// TIA Portal V17 export
// export: Created 2023-02-13T11:16:52.2273647Z, ExportSetting WithDefaults, DisplayName Totally Integrated Automation Portal, DisplayVersion V17, DisplayName TIA Portal Openness, DisplayVersion V17, DisplayName TIA Portal Teamcenter Gateway, DisplayVersion V17, DisplayName TIA Portal Version Control Interface, DisplayVersion V17, DisplayName SINAMICS Startdrive Advanced, DisplayVersion V17, DisplayName SINAMICS Startdrive G130, G150, S120, S150, SINAMICS MV, S210, DisplayVersion V17, DisplayName SINAMICS Startdrive G110M, G120, G120C, G120D, G120P, G115D, DisplayVersion V17, DisplayName STEP 7 Professional, DisplayVersion V17, DisplayName STEP 7 Safety, DisplayVersion V17, DisplayName WinCC Professional, DisplayVersion V17
FUNCTION_BLOCK "HWT"   // FB350, LAD
{ S7_Optimized_Access := 'TRUE' }
VERSION : 0.1
// stored: AutoNumber false, IsIECCheckEnabled false, IsRetainMemResEnabled false, MemoryReserve 100, SetENOAutomatically false, UDAEnableTagReadback false
   VAR_INPUT
      "IN_FBAV.01" : Bool := FALSE;   // Tank Return Valve
      "IN_FBAV.02" : Bool := FALSE;   // Tank Water Inlet Valve
      "IN_FBAV.03" : Bool := FALSE;   // Tank CIP Return Valve
      "IN_FBAV.04" : Bool := FALSE;   // Tank CIP Inlet Valve
      "IN_FBAV.10" : Bool := FALSE;   // Steam Shutoff Valve
      "IN_FBCV.10" : Bool := FALSE;   // Steam Control Valve
      "IN_FS.01" : Bool := FALSE;   // Line Flow Switch
      IN_LT01 : Real;   // Tank Level Transmitter
      IN_TT01 : Real;   // Tank Temp. Transmitter
      IN_TT02 : Real;   // Line Temp. Transmitter
      "IN_FBP.01" : Bool;   // Hot Water Pump
      "IN_P.01-Speed" : Real := 0.0;   // Hot Water Pump AV Speed
      DosePumpSpeed : Real;
      "DoseON-OFF" : Bool;
      "DosePumpON-OFF" : Bool;
      CIPPulse : Bool;
      Line_OK : Bool;
   END_VAR
   VAR_OUTPUT
      "OUT_AV.01" : Bool := FALSE;   // Tank Return Valve
      "OUT_AV.02" : Bool := FALSE;   // Tank Water Inlet Valve
      "OUT_AV.03" : Bool := FALSE;   // Tank CIP Return Valve
      "OUT_AV.04" : Bool := FALSE;   // Tank CIP Inlet Valve
      "OUT_AV.10" : Bool := FALSE;   // Steam Shutoff Valve
      "OUT_CV.10" : Bool := FALSE;   // Steam Control Valve
      Q_PID_Setpoint : Real;
      Q_PID_PV_IN : Real;
      "OUT_FS.01" : Bool := FALSE;   // Line Flow Switch
      "OUT_LT.01" : Real;   // Tank Level Transmitter
      "OUT_TT.01" : Real;   // Tank Temp. Transmitter
      "OUT_TT.02" : Real;   // Line Temp. Transmitter
      "OUT_P.01" : Bool := FALSE;   // Hot Water Pump
      "OUT_P.01-Speed" : Real := 0.0;   // Hot Water Pump SP Speed
      OUT_CIP_Request : Bool;
      Q_WH_Tank_Ready : Bool;
   END_VAR
   VAR
      Cmd : Struct
         Start_Prosses : Bool;
         Start_Preheat : Bool;
         HWT_Mode : Bool;
         Ready_for_Mix : Bool;
         "CIP Request" : Bool;
         Pump_Mode : Bool;
         Pump_Man_ON_OFF : Bool;
      END_STRUCT;
      Param : Struct
         SP_Level_LL : Real := 10.0;
         SP_Level_ML : Real := 80.0;
         SP_Level_HL : Real := 100.0;
         SP_Temp_Prepar : Real := 80.0;
         SP_Temp_Process : Real := 80.0;
         SP_PumpSpeed : Real := 80.0;
         L_Hi_Lim : Real := 100.0;
         L_Lo_Lim : Real := 0.0;
         L_Hys : Real := 5.0;
         T_Hi_Lim : Real := 100.0;
         T_Lo_Lim : Real := 0.0;
         T_Hys : Real := 2.0;
         CIP_Ret_ON_SP : Real := 5.0;
         CIP_Ret_OFF_SP : Real;
      END_STRUCT;
      State : Struct
         Tank_LL : Bool;
         Tank_ML : Bool;
         Tank_HL : Bool;
         Temp_Preheat_OK : Bool;
         Temp_Process_OK : Bool;
         Tank_Heating : Bool;
         "Tank is Ready" : Bool;
         "Tank in transfer" : Bool;
         Enable_WHT_Mode : Bool;
         Enable_Ready : Bool;
         Ready_for_Mix : Bool;
         "CIP Request Enable" : Bool;
         "Tank in CIP" : Bool;
         CIP_Request_OK : Bool;
         CIP_ReturnON : Bool;
         HWT_Status : Int;
         Temp_Actual : Real;
      END_STRUCT;
      L_Hys_Abs : Real;
      T_Hys_Abs : Real;
      Hys_Level_HL : Real;
      Hys_Level_ML : Real;
      Hys_Level_LL : Real;
      "Hys SP_SP_Prepar" : Real;
      "Hys SP_SP_Process" : Real;
      "Hys SP_SP_" : Real;
      alwaysON : Bool;
      r : Struct
         PosE1 : Bool;
         PosE2 : Bool;
         PosE3 : Bool;
         PosE4 : Bool;
         PosE5 : Bool;
         PosE6 : Bool;
         PosE7 : Bool;
         PosE8 : Bool;
         PosE9 : Bool;
         PosE10 : Bool;
         PosE11 : Bool;
         PosE12 : Bool;
         PosE13 : Bool;
         PosE14 : Bool;
         PosE15 : Bool;
         PosE16 : Bool;
         PosE17 : Bool;
         PosE18 : Bool;
         PosE19 : Bool;
         PosE20 : Bool;
         PosE21 : Bool;
         PosE22 : Bool;
         PosE23 : Bool;
         PosE24 : Bool;
         PosE25 : Bool;
         PosE26 : Bool;
         PosE27 : Bool;
         PosE28 : Bool;
         PosE29 : Bool;
         PosE30 : Bool;
         PosE31 : Bool;
         PosE32 : Bool;
      END_STRUCT;
      Actuator : Struct
         AV_Inlet : Bool;
         AV_Return : Bool;
         CV_Steam : Bool;
         Pump : Bool;
      END_STRUCT;
      r_Pump : Bool;
      r_PumpTim { S7_SetPoint := 'True'} : IEC_TIMER;
      Alarm : Word;
      Event : Word;
   END_VAR
   VAR_TEMP   // added for the SCL form of the ladder/FBD networks
      _w1 : Bool;
      _w2 : Bool;
   END_VAR
BEGIN

REGION Network 1: Always_ON
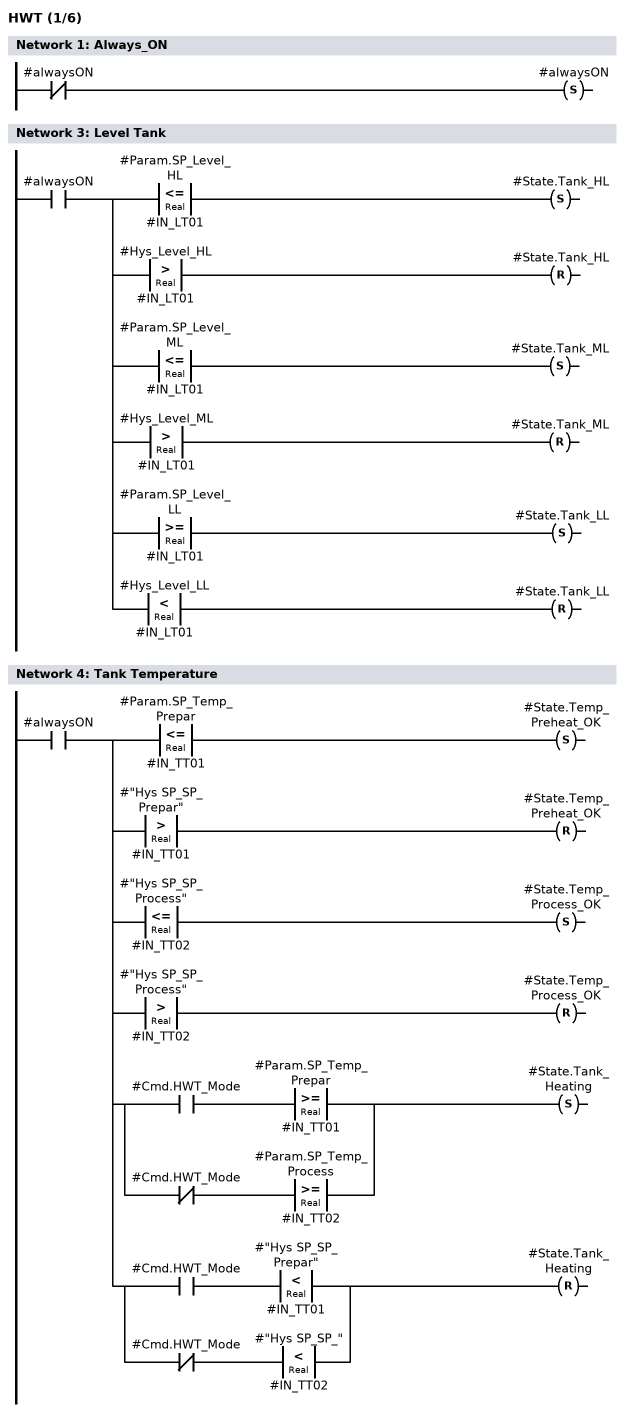
   RUNG wire#powerrail
      I_Contact( #alwaysON )
      S_Coil( #alwaysON )
   END_RUNG
   // the same network as SCL:
   IF NOT #alwaysON THEN #alwaysON := TRUE; END_IF;
END_REGION

NETWORK
TITLE = Hys Calculation
//Level Hys Absolute
      L     #Param.L_Hi_Lim;
      L     #Param.L_Lo_Lim;
      -R;
      L     100.0;
      /R;
      L     #Param.L_Hys;
      *R;
      T     #L_Hys_Abs;
//Temp. Hys Absolute
      L     #Param.T_Hi_Lim;
      L     #Param.T_Lo_Lim;
      -R;
      L     100.0;
      /R;
      L     #Param.T_Hys;
      *R;
      T     #T_Hys_Abs;
//Tank High Level
      L     #Param.SP_Level_HL;
      L     #L_Hys_Abs;
      -R;
      T     #Hys_Level_HL;
//Tank Mid Level
      L     #Param.SP_Level_ML;
      L     #L_Hys_Abs;
      -R;
      T     #Hys_Level_ML;
//Tank Low Level
      L     #Param.SP_Level_LL;
      L     #L_Hys_Abs;
      +R;
      T     #Hys_Level_LL;
//Temp. Preheat Hys
      L     #Param.SP_Temp_Prepar;
      L     #T_Hys_Abs;
      +R;
      T     #"Hys SP_SP_Prepar";
//Temp. Transfer Hys
      L     #Param.SP_Temp_Process;
      L     #T_Hys_Abs;
      -R;
      T     #"Hys SP_SP_Process";
//Temp. Transfer Heating Hys
      L     #Param.SP_Temp_Process;
      L     #T_Hys_Abs;
      +R;
      T     #"Hys SP_SP_";


REGION Network 3: Level Tank
   RUNG wire#powerrail
      Contact( #alwaysON )
      wire#w1
      { S7_Templates := "SrcType := Real" } LE_Contact(in1 := #Param.SP_Level_HL, in2 := #IN_LT01)
      S_Coil( #State.Tank_HL )
   END_RUNG
   RUNG wire#w1
      { S7_Templates := "SrcType := Real" } GT_Contact(in1 := #Hys_Level_HL, in2 := #IN_LT01)
      R_Coil( #State.Tank_HL )
   END_RUNG
   RUNG wire#w1
      { S7_Templates := "SrcType := Real" } LE_Contact(in1 := #Param.SP_Level_ML, in2 := #IN_LT01)
      S_Coil( #State.Tank_ML )
   END_RUNG
   RUNG wire#w1
      { S7_Templates := "SrcType := Real" } GT_Contact(in1 := #Hys_Level_ML, in2 := #IN_LT01)
      R_Coil( #State.Tank_ML )
   END_RUNG
   RUNG wire#w1
      { S7_Templates := "SrcType := Real" } GE_Contact(in1 := #Param.SP_Level_LL, in2 := #IN_LT01)
      S_Coil( #State.Tank_LL )
   END_RUNG
   RUNG wire#w1
      { S7_Templates := "SrcType := Real" } LT_Contact(in1 := #Hys_Level_LL, in2 := #IN_LT01)
      R_Coil( #State.Tank_LL )
   END_RUNG
   // the same network as SCL:
   IF #alwaysON AND (#Param.SP_Level_HL <= #IN_LT01) THEN #State.Tank_HL := TRUE; END_IF;
   IF #alwaysON AND (#Hys_Level_HL > #IN_LT01) THEN #State.Tank_HL := FALSE; END_IF;
   IF #alwaysON AND (#Param.SP_Level_ML <= #IN_LT01) THEN #State.Tank_ML := TRUE; END_IF;
   IF #alwaysON AND (#Hys_Level_ML > #IN_LT01) THEN #State.Tank_ML := FALSE; END_IF;
   IF #alwaysON AND (#Param.SP_Level_LL >= #IN_LT01) THEN #State.Tank_LL := TRUE; END_IF;
   IF #alwaysON AND (#Hys_Level_LL < #IN_LT01) THEN #State.Tank_LL := FALSE; END_IF;
END_REGION

REGION Network 4: Tank Temperature
   RUNG wire#powerrail
      Contact( #alwaysON )
      wire#w1
      { S7_Templates := "SrcType := Real" } LE_Contact(in1 := #Param.SP_Temp_Prepar, in2 := #IN_TT01)
      S_Coil( #State.Temp_Preheat_OK )
   END_RUNG
   RUNG wire#w1
      { S7_Templates := "SrcType := Real" } GT_Contact(in1 := #"Hys SP_SP_Prepar", in2 := #IN_TT01)
      R_Coil( #State.Temp_Preheat_OK )
   END_RUNG
   RUNG wire#w1
      { S7_Templates := "SrcType := Real" } LE_Contact(in1 := #"Hys SP_SP_Process", in2 := #IN_TT02)
      S_Coil( #State.Temp_Process_OK )
   END_RUNG
   RUNG wire#w1
      { S7_Templates := "SrcType := Real" } GT_Contact(in1 := #"Hys SP_SP_Process", in2 := #IN_TT02)
      R_Coil( #State.Temp_Process_OK )
   END_RUNG
   RUNG wire#w1
      Contact( #Cmd.HWT_Mode )
      { S7_Templates := "SrcType := Real" } GE_Contact(in1 := #Param.SP_Temp_Prepar, in2 := #IN_TT01)
      wire#w2
      S_Coil( #State.Tank_Heating )
   END_RUNG
   RUNG wire#w1
      I_Contact( #Cmd.HWT_Mode )
      { S7_Templates := "SrcType := Real" } GE_Contact(in1 := #Param.SP_Temp_Process, in2 := #IN_TT02)
   END_RUNG wire#w2
   RUNG wire#w1
      Contact( #Cmd.HWT_Mode )
      { S7_Templates := "SrcType := Real" } LT_Contact(in1 := #"Hys SP_SP_Prepar", in2 := #IN_TT01)
      wire#w3
      R_Coil( #State.Tank_Heating )
   END_RUNG
   RUNG wire#w1
      I_Contact( #Cmd.HWT_Mode )
      { S7_Templates := "SrcType := Real" } LT_Contact(in1 := #"Hys SP_SP_", in2 := #IN_TT02)
   END_RUNG wire#w3
   // the same network as SCL:
   IF #alwaysON AND (#Param.SP_Temp_Prepar <= #IN_TT01) THEN #State.Temp_Preheat_OK := TRUE; END_IF;
   IF #alwaysON AND (#"Hys SP_SP_Prepar" > #IN_TT01) THEN #State.Temp_Preheat_OK := FALSE; END_IF;
   IF #alwaysON AND (#"Hys SP_SP_Process" <= #IN_TT02) THEN #State.Temp_Process_OK := TRUE; END_IF;
   IF #alwaysON AND (#"Hys SP_SP_Process" > #IN_TT02) THEN #State.Temp_Process_OK := FALSE; END_IF;
   IF #alwaysON AND ((#Cmd.HWT_Mode AND (#Param.SP_Temp_Prepar >= #IN_TT01)) OR (NOT #Cmd.HWT_Mode AND (#Param.SP_Temp_Process >= #IN_TT02))) THEN
       #State.Tank_Heating := TRUE;
   END_IF;
   IF #alwaysON AND ((#Cmd.HWT_Mode AND (#"Hys SP_SP_Prepar" < #IN_TT01)) OR (NOT #Cmd.HWT_Mode AND (#"Hys SP_SP_" < #IN_TT02))) THEN
       #State.Tank_Heating := FALSE;
   END_IF;
END_REGION

REGION Network 5: Reset Command
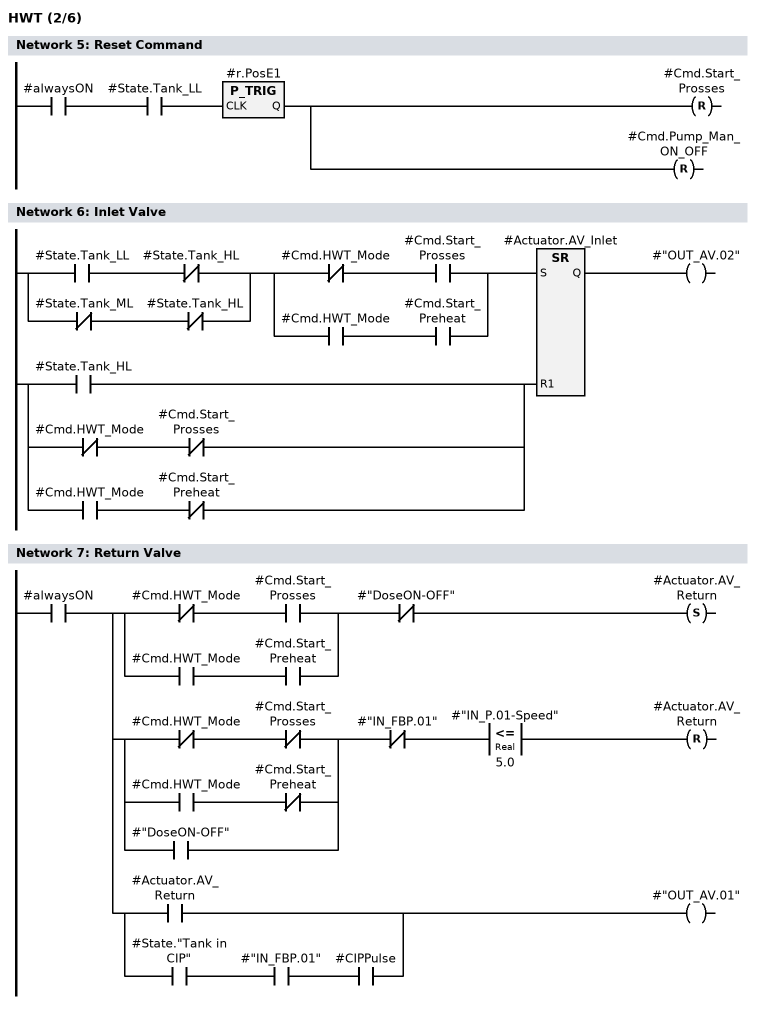
   RUNG wire#powerrail
      Contact( #alwaysON )
      Contact( #State.Tank_LL )
      P_Trig( #r.PosE1 )
      wire#w1
      R_Coil( #Cmd.Start_Prosses )
   END_RUNG
   RUNG wire#w1
      R_Coil( #Cmd.Pump_Man_ON_OFF )
   END_RUNG
   // the same network as SCL:
   #_w1 := #alwaysON AND #State.Tank_LL;
   #_w2 := #_w1 AND NOT #r.PosE1;   // rising edge
   #r.PosE1 := #_w1;
   IF #_w2 THEN
       #Cmd.Start_Prosses := FALSE;
       #Cmd.Pump_Man_ON_OFF := FALSE;
   END_IF;
END_REGION

REGION Network 6: Inlet Valve
   RUNG wire#powerrail
      Contact( #State.Tank_LL )
      I_Contact( #State.Tank_HL )
      wire#w1
      I_Contact( #Cmd.HWT_Mode )
      Contact( #Cmd.Start_Prosses )
      wire#w2
      S_SR(operand := #Actuator.AV_Inlet, r1 := wire#w3)
      Coil( #"OUT_AV.02" )
   END_RUNG
   RUNG wire#powerrail
      I_Contact( #State.Tank_ML )
      I_Contact( #State.Tank_HL )
   END_RUNG wire#w1
   RUNG wire#w1
      Contact( #Cmd.HWT_Mode )
      Contact( #Cmd.Start_Preheat )
   END_RUNG wire#w2
   RUNG wire#powerrail
      Contact( #State.Tank_HL )
   END_RUNG wire#w3
   RUNG wire#powerrail
      I_Contact( #Cmd.HWT_Mode )
      I_Contact( #Cmd.Start_Prosses )
   END_RUNG wire#w3
   RUNG wire#powerrail
      Contact( #Cmd.HWT_Mode )
      I_Contact( #Cmd.Start_Preheat )
   END_RUNG wire#w3
   // the same network as SCL:
   IF ((#State.Tank_LL AND NOT #State.Tank_HL) OR (NOT #State.Tank_ML AND NOT #State.Tank_HL)) AND ((NOT #Cmd.HWT_Mode AND #Cmd.Start_Prosses) OR (#Cmd.HWT_Mode AND #Cmd.Start_Preheat)) THEN
       #Actuator.AV_Inlet := TRUE;   // SR flip-flop
   END_IF;
   IF #State.Tank_HL OR (NOT #Cmd.HWT_Mode AND NOT #Cmd.Start_Prosses) OR (#Cmd.HWT_Mode AND NOT #Cmd.Start_Preheat) THEN
       #Actuator.AV_Inlet := FALSE;
   END_IF;
   #"OUT_AV.02" := #Actuator.AV_Inlet;
END_REGION

REGION Network 7: Return Valve
   RUNG wire#powerrail
      Contact( #alwaysON )
      wire#w1
      I_Contact( #Cmd.HWT_Mode )
      Contact( #Cmd.Start_Prosses )
      wire#w2
      I_Contact( #"DoseON-OFF" )
      S_Coil( #Actuator.AV_Return )
   END_RUNG
   RUNG wire#w1
      Contact( #Cmd.HWT_Mode )
      Contact( #Cmd.Start_Preheat )
   END_RUNG wire#w2
   RUNG wire#w1
      I_Contact( #Cmd.HWT_Mode )
      I_Contact( #Cmd.Start_Prosses )
      wire#w3
      I_Contact( #"IN_FBP.01" )
      { S7_Templates := "SrcType := Real" } LE_Contact(in1 := #"IN_P.01-Speed", in2 := 5.0)
      R_Coil( #Actuator.AV_Return )
   END_RUNG
   RUNG wire#w1
      Contact( #Cmd.HWT_Mode )
      I_Contact( #Cmd.Start_Preheat )
   END_RUNG wire#w3
   RUNG wire#w1
      Contact( #"DoseON-OFF" )
   END_RUNG wire#w3
   RUNG wire#w1
      Contact( #Actuator.AV_Return )
      wire#w4
      Coil( #"OUT_AV.01" )
   END_RUNG
   RUNG wire#w1
      Contact( #State."Tank in CIP" )
      Contact( #"IN_FBP.01" )
      Contact( #CIPPulse )
   END_RUNG wire#w4
   // the same network as SCL:
   IF #alwaysON AND ((NOT #Cmd.HWT_Mode AND #Cmd.Start_Prosses) OR (#Cmd.HWT_Mode AND #Cmd.Start_Preheat)) AND NOT #"DoseON-OFF" THEN
       #Actuator.AV_Return := TRUE;
   END_IF;
   IF #alwaysON AND ((NOT #Cmd.HWT_Mode AND NOT #Cmd.Start_Prosses) OR (#Cmd.HWT_Mode AND NOT #Cmd.Start_Preheat) OR #"DoseON-OFF") AND NOT #"IN_FBP.01" AND (#"IN_P.01-Speed" <= 5.0) THEN
       #Actuator.AV_Return := FALSE;
   END_IF;
   #"OUT_AV.01" := #alwaysON AND (#Actuator.AV_Return OR (#State."Tank in CIP" AND #"IN_FBP.01" AND #CIPPulse));
END_REGION

REGION Network 8: Pump HW-Supply
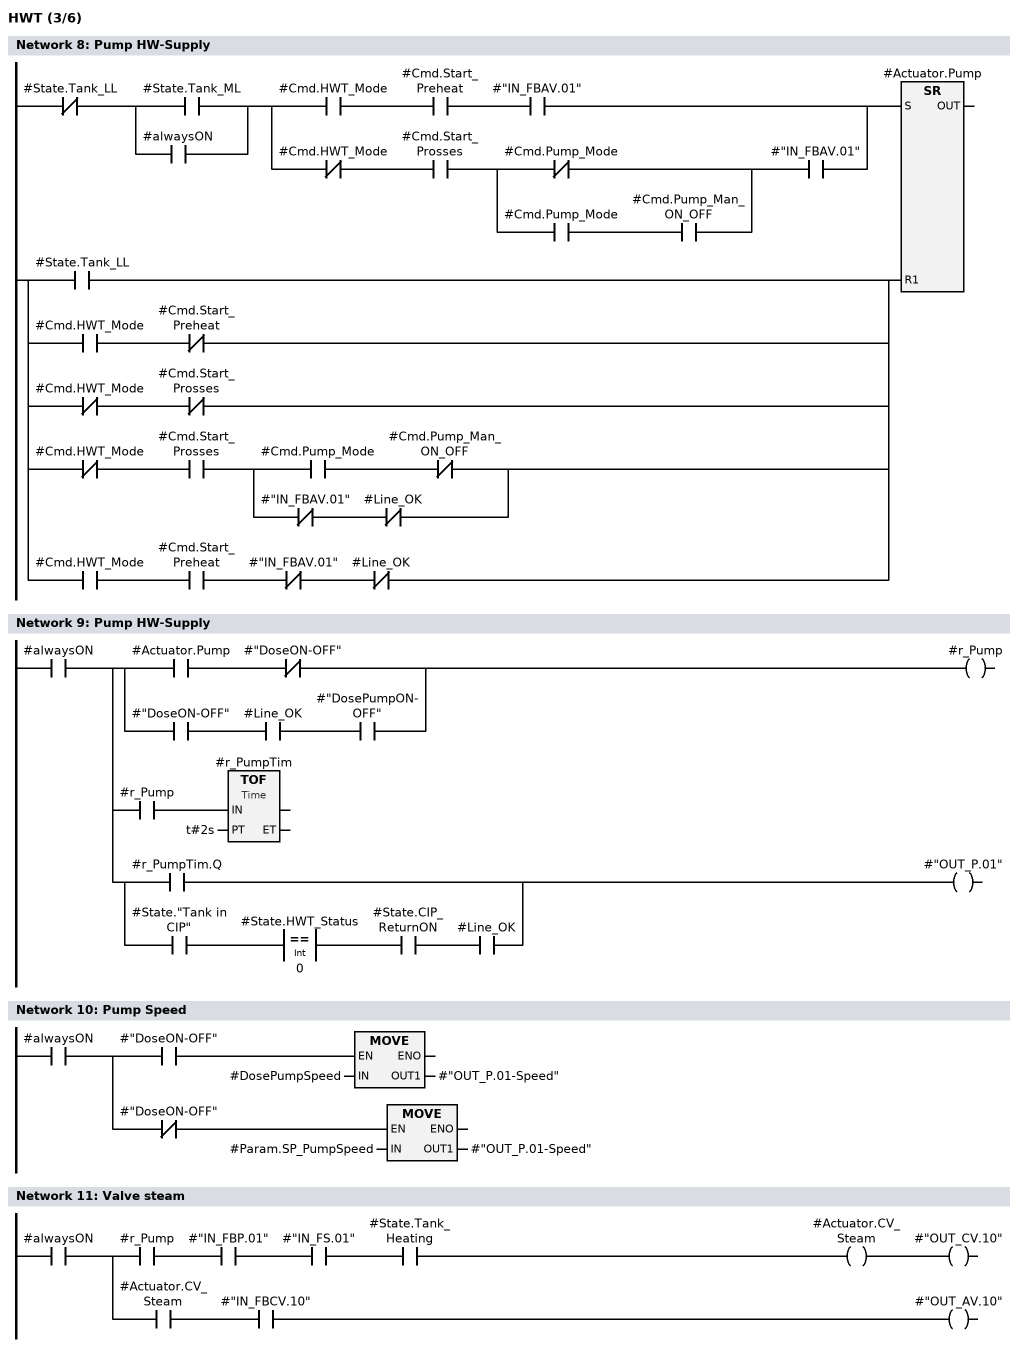
   RUNG wire#powerrail
      I_Contact( #State.Tank_LL )
      wire#w1
      Contact( #State.Tank_ML )
      wire#w2
      Contact( #Cmd.HWT_Mode )
      Contact( #Cmd.Start_Preheat )
      Contact( #"IN_FBAV.01" )
      wire#w3
      S_SR(operand := #Actuator.Pump, r1 := wire#w7)
   END_RUNG
   RUNG wire#w1
      Contact( #alwaysON )
   END_RUNG wire#w2
   RUNG wire#w2
      I_Contact( #Cmd.HWT_Mode )
      Contact( #Cmd.Start_Prosses )
      wire#w4
      I_Contact( #Cmd.Pump_Mode )
      wire#w5
      Contact( #"IN_FBAV.01" )
   END_RUNG wire#w3
   RUNG wire#w4
      Contact( #Cmd.Pump_Mode )
      Contact( #Cmd.Pump_Man_ON_OFF )
   END_RUNG wire#w5
   RUNG wire#powerrail
      Contact( #State.Tank_LL )
   END_RUNG wire#w7
   RUNG wire#powerrail
      Contact( #Cmd.HWT_Mode )
      I_Contact( #Cmd.Start_Preheat )
   END_RUNG wire#w7
   RUNG wire#powerrail
      I_Contact( #Cmd.HWT_Mode )
      I_Contact( #Cmd.Start_Prosses )
   END_RUNG wire#w7
   RUNG wire#powerrail
      I_Contact( #Cmd.HWT_Mode )
      Contact( #Cmd.Start_Prosses )
      wire#w6
      Contact( #Cmd.Pump_Mode )
      I_Contact( #Cmd.Pump_Man_ON_OFF )
   END_RUNG wire#w7
   RUNG wire#w6
      I_Contact( #"IN_FBAV.01" )
      I_Contact( #Line_OK )
   END_RUNG wire#w7
   RUNG wire#powerrail
      Contact( #Cmd.HWT_Mode )
      Contact( #Cmd.Start_Preheat )
      I_Contact( #"IN_FBAV.01" )
      I_Contact( #Line_OK )
   END_RUNG wire#w7
   // the same network as SCL:
   IF NOT #State.Tank_LL AND (#State.Tank_ML OR #alwaysON) AND ((#Cmd.HWT_Mode AND #Cmd.Start_Preheat AND #"IN_FBAV.01") OR (NOT #Cmd.HWT_Mode AND #Cmd.Start_Prosses AND (NOT #Cmd.Pump_Mode OR (#Cmd.Pump_Mode AND #Cmd.Pump_Man_ON_OFF)) AND #"IN_FBAV.01")) THEN
       #Actuator.Pump := TRUE;   // SR flip-flop
   END_IF;
   IF #State.Tank_LL OR (#Cmd.HWT_Mode AND NOT #Cmd.Start_Preheat) OR (NOT #Cmd.HWT_Mode AND NOT #Cmd.Start_Prosses) OR (NOT #Cmd.HWT_Mode AND #Cmd.Start_Prosses AND ((#Cmd.Pump_Mode AND NOT #Cmd.Pump_Man_ON_OFF) OR (NOT #"IN_FBAV.01" AND NOT #Line_OK))) OR (#Cmd.HWT_Mode AND #Cmd.Start_Preheat AND NOT #"IN_FBAV.01" AND NOT #Line_OK) THEN
       #Actuator.Pump := FALSE;
   END_IF;
END_REGION

REGION Network 9: Pump HW-Supply
   RUNG wire#powerrail
      Contact( #alwaysON )
      wire#w1
      Contact( #Actuator.Pump )
      I_Contact( #"DoseON-OFF" )
      wire#w2
      Coil( #r_Pump )
   END_RUNG
   RUNG wire#w1
      Contact( #"DoseON-OFF" )
      Contact( #Line_OK )
      Contact( #"DosePumpON-OFF" )
   END_RUNG wire#w2
   RUNG wire#w1
      Contact( #r_Pump )
      { S7_Templates := "time_type := Time" } #r_PumpTim.TOF(pt := t#2s, et =>)
   END_RUNG
   RUNG wire#w1
      Contact( #r_PumpTim.Q )
      wire#w3
      Coil( #"OUT_P.01" )
   END_RUNG
   RUNG wire#w1
      Contact( #State."Tank in CIP" )
      { S7_Templates := "SrcType := Int" } EQ_Contact(in1 := #State.HWT_Status, in2 := 0)
      Contact( #State.CIP_ReturnON )
      Contact( #Line_OK )
   END_RUNG wire#w3
   // the same network as SCL:
   #r_Pump := #alwaysON AND ((#Actuator.Pump AND NOT #"DoseON-OFF") OR (#"DoseON-OFF" AND #Line_OK AND #"DosePumpON-OFF"));
   #r_PumpTim.TOF(IN := #alwaysON AND #r_Pump, PT := t#2s);
   #"OUT_P.01" := #alwaysON AND (#r_PumpTim.Q OR (#State."Tank in CIP" AND (#State.HWT_Status = 0) AND #State.CIP_ReturnON AND #Line_OK));
END_REGION

REGION Network 10: Pump Speed
   RUNG wire#powerrail
      Contact( #alwaysON )
      wire#w1
      Contact( #"DoseON-OFF" )
      Move(in := #DosePumpSpeed, out1 => #"OUT_P.01-Speed")
   END_RUNG
   RUNG wire#w1
      I_Contact( #"DoseON-OFF" )
      Move(in := #Param.SP_PumpSpeed, out1 => #"OUT_P.01-Speed")
   END_RUNG
   // the same network as SCL:
   IF #alwaysON AND #"DoseON-OFF" THEN #"OUT_P.01-Speed" := #DosePumpSpeed; END_IF;
   IF #alwaysON AND NOT #"DoseON-OFF" THEN #"OUT_P.01-Speed" := #Param.SP_PumpSpeed; END_IF;
END_REGION

REGION Network 11: Valve steam
   RUNG wire#powerrail
      Contact( #alwaysON )
      wire#w1
      Contact( #r_Pump )
      Contact( #"IN_FBP.01" )
      Contact( #"IN_FS.01" )
      Contact( #State.Tank_Heating )
      Coil( #Actuator.CV_Steam )
      Coil( #"OUT_CV.10" )
   END_RUNG
   RUNG wire#w1
      Contact( #Actuator.CV_Steam )
      Contact( #"IN_FBCV.10" )
      Coil( #"OUT_AV.10" )
   END_RUNG
   // the same network as SCL:
   #Actuator.CV_Steam := #alwaysON AND #r_Pump AND #"IN_FBP.01" AND #"IN_FS.01" AND #State.Tank_Heating;
   #"OUT_CV.10" := #Actuator.CV_Steam;
   #"OUT_AV.10" := #alwaysON AND #Actuator.CV_Steam AND #"IN_FBCV.10";
END_REGION

REGION Network 12: PID Setpoint Preparation
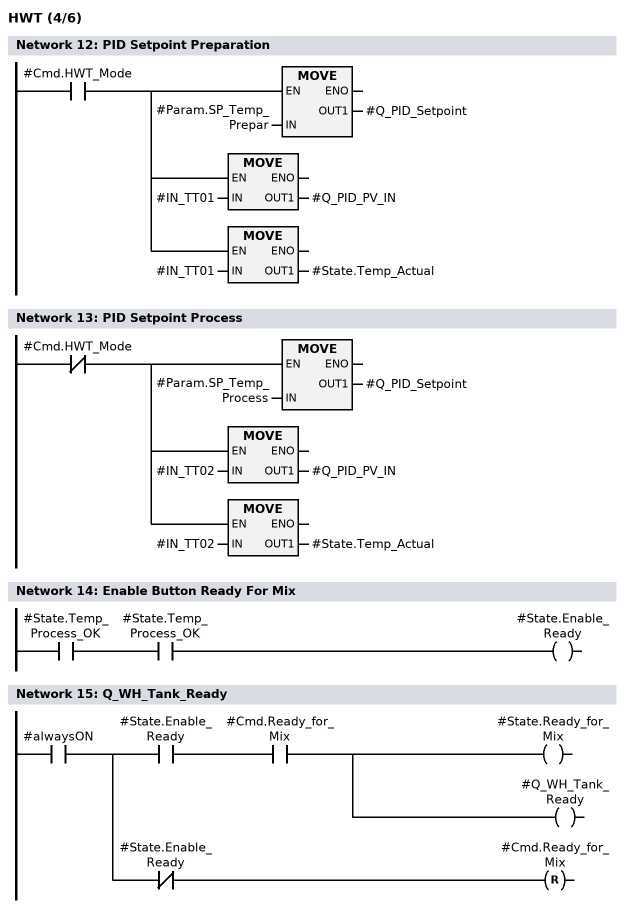
   RUNG wire#powerrail
      Contact( #Cmd.HWT_Mode )
      wire#w1
      { S7_GenerateENO := "TRUE" } Move(in := #Param.SP_Temp_Prepar, out1 => #Q_PID_Setpoint)
   END_RUNG
   RUNG wire#w1
      { S7_GenerateENO := "TRUE" } Move(in := #IN_TT01, out1 => #Q_PID_PV_IN)
   END_RUNG
   RUNG wire#w1
      { S7_GenerateENO := "TRUE" } Move(in := #IN_TT01, out1 => #State.Temp_Actual)
   END_RUNG
   // the same network as SCL:
   IF #Cmd.HWT_Mode THEN
       #Q_PID_Setpoint := #Param.SP_Temp_Prepar;
       #Q_PID_PV_IN := #IN_TT01;
       #State.Temp_Actual := #IN_TT01;
   END_IF;
END_REGION

REGION Network 13: PID Setpoint Process
   RUNG wire#powerrail
      I_Contact( #Cmd.HWT_Mode )
      wire#w1
      { S7_GenerateENO := "TRUE" } Move(in := #Param.SP_Temp_Process, out1 => #Q_PID_Setpoint)
   END_RUNG
   RUNG wire#w1
      { S7_GenerateENO := "TRUE" } Move(in := #IN_TT02, out1 => #Q_PID_PV_IN)
   END_RUNG
   RUNG wire#w1
      { S7_GenerateENO := "TRUE" } Move(in := #IN_TT02, out1 => #State.Temp_Actual)
   END_RUNG
   // the same network as SCL:
   IF NOT #Cmd.HWT_Mode THEN
       #Q_PID_Setpoint := #Param.SP_Temp_Process;
       #Q_PID_PV_IN := #IN_TT02;
       #State.Temp_Actual := #IN_TT02;
   END_IF;
END_REGION

REGION Network 14: Enable Button Ready For Mix
   RUNG wire#powerrail
      Contact( #State.Temp_Process_OK )
      Contact( #State.Temp_Process_OK )
      Coil( #State.Enable_Ready )
   END_RUNG
   // the same network as SCL:
   #State.Enable_Ready := #State.Temp_Process_OK AND #State.Temp_Process_OK;
END_REGION

REGION Network 15: Q_WH_Tank_Ready
   RUNG wire#powerrail
      Contact( #alwaysON )
      wire#w1
      Contact( #State.Enable_Ready )
      Contact( #Cmd.Ready_for_Mix )
      wire#w2
      Coil( #State.Ready_for_Mix )
   END_RUNG
   RUNG wire#w2
      Coil( #Q_WH_Tank_Ready )
   END_RUNG
   RUNG wire#w1
      I_Contact( #State.Enable_Ready )
      R_Coil( #Cmd.Ready_for_Mix )
   END_RUNG
   // the same network as SCL:
   #State.Ready_for_Mix := #alwaysON AND #State.Enable_Ready AND #Cmd.Ready_for_Mix;
   #Q_WH_Tank_Ready := #State.Ready_for_Mix;
   IF #alwaysON AND NOT #State.Enable_Ready THEN #Cmd.Ready_for_Mix := FALSE; END_IF;
END_REGION

REGION Network 16: CIP
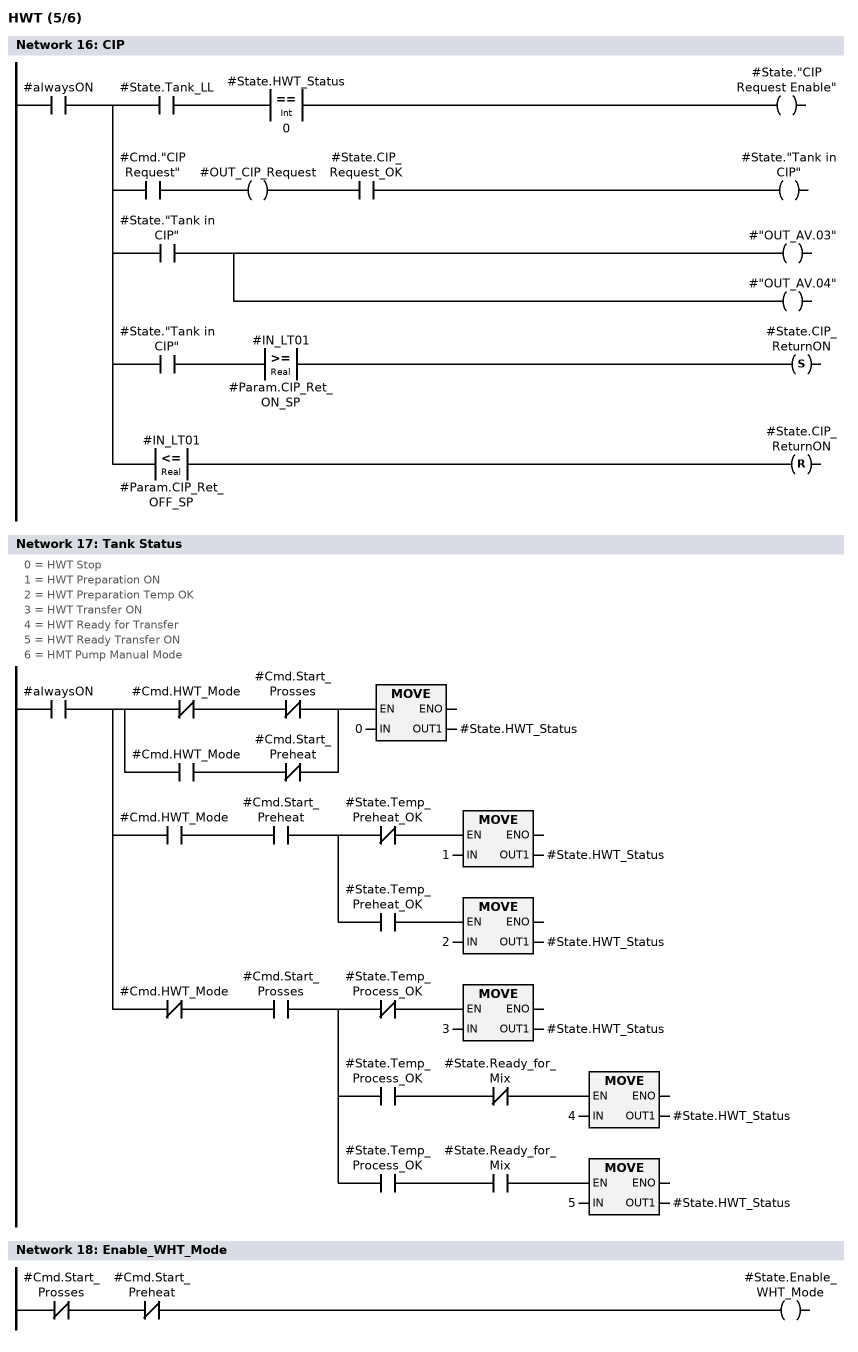
   RUNG wire#powerrail
      Contact( #alwaysON )
      wire#w1
      Contact( #State.Tank_LL )
      { S7_Templates := "SrcType := Int" } EQ_Contact(in1 := #State.HWT_Status, in2 := 0)
      Coil( #State."CIP Request Enable" )
   END_RUNG
   RUNG wire#w1
      Contact( #Cmd."CIP Request" )
      Coil( #OUT_CIP_Request )
      Contact( #State.CIP_Request_OK )
      Coil( #State."Tank in CIP" )
   END_RUNG
   RUNG wire#w1
      Contact( #State."Tank in CIP" )
      wire#w2
      Coil( #"OUT_AV.03" )
   END_RUNG
   RUNG wire#w2
      Coil( #"OUT_AV.04" )
   END_RUNG
   RUNG wire#w1
      Contact( #State."Tank in CIP" )
      { S7_Templates := "SrcType := Real" } GE_Contact(in1 := #IN_LT01, in2 := #Param.CIP_Ret_ON_SP)
      S_Coil( #State.CIP_ReturnON )
   END_RUNG
   RUNG wire#w1
      { S7_Templates := "SrcType := Real" } LE_Contact(in1 := #IN_LT01, in2 := #Param.CIP_Ret_OFF_SP)
      R_Coil( #State.CIP_ReturnON )
   END_RUNG
   // the same network as SCL:
   #State."CIP Request Enable" := #alwaysON AND #State.Tank_LL AND (#State.HWT_Status = 0);
   #OUT_CIP_Request := #alwaysON AND #Cmd."CIP Request";
   #State."Tank in CIP" := #OUT_CIP_Request AND #State.CIP_Request_OK;
   #"OUT_AV.03" := #alwaysON AND #State."Tank in CIP";
   #"OUT_AV.04" := #"OUT_AV.03";
   IF #alwaysON AND #State."Tank in CIP" AND (#IN_LT01 >= #Param.CIP_Ret_ON_SP) THEN
       #State.CIP_ReturnON := TRUE;
   END_IF;
   IF #alwaysON AND (#IN_LT01 <= #Param.CIP_Ret_OFF_SP) THEN #State.CIP_ReturnON := FALSE; END_IF;
END_REGION

REGION Network 17: Tank Status
   // 0 = HWT Stop
   // 1 = HWT Preparation ON
   // 2 = HWT Preparation Temp OK
   // 3 = HWT Transfer ON
   // 4 = HWT Ready for Transfer
   // 5 = HWT Ready Transfer ON
   // 6 = HMT Pump Manual Mode
   RUNG wire#powerrail
      Contact( #alwaysON )
      wire#w1
      I_Contact( #Cmd.HWT_Mode )
      I_Contact( #Cmd.Start_Prosses )
      wire#w2
      { S7_GenerateENO := "TRUE" } Move(in := 0, out1 => #State.HWT_Status)
   END_RUNG
   RUNG wire#w1
      Contact( #Cmd.HWT_Mode )
      I_Contact( #Cmd.Start_Preheat )
   END_RUNG wire#w2
   RUNG wire#w1
      Contact( #Cmd.HWT_Mode )
      Contact( #Cmd.Start_Preheat )
      wire#w3
      I_Contact( #State.Temp_Preheat_OK )
      { S7_GenerateENO := "TRUE" } Move(in := 1, out1 => #State.HWT_Status)
   END_RUNG
   RUNG wire#w3
      Contact( #State.Temp_Preheat_OK )
      { S7_GenerateENO := "TRUE" } Move(in := 2, out1 => #State.HWT_Status)
   END_RUNG
   RUNG wire#w1
      I_Contact( #Cmd.HWT_Mode )
      Contact( #Cmd.Start_Prosses )
      wire#w4
      I_Contact( #State.Temp_Process_OK )
      { S7_GenerateENO := "TRUE" } Move(in := 3, out1 => #State.HWT_Status)
   END_RUNG
   RUNG wire#w4
      Contact( #State.Temp_Process_OK )
      I_Contact( #State.Ready_for_Mix )
      { S7_GenerateENO := "TRUE" } Move(in := 4, out1 => #State.HWT_Status)
   END_RUNG
   RUNG wire#w4
      Contact( #State.Temp_Process_OK )
      Contact( #State.Ready_for_Mix )
      { S7_GenerateENO := "TRUE" } Move(in := 5, out1 => #State.HWT_Status)
   END_RUNG
   // the same network as SCL:
   IF #alwaysON AND ((NOT #Cmd.HWT_Mode AND NOT #Cmd.Start_Prosses) OR (#Cmd.HWT_Mode AND NOT #Cmd.Start_Preheat)) THEN
       #State.HWT_Status := 0;
   END_IF;
   #_w1 := #alwaysON AND #Cmd.HWT_Mode AND #Cmd.Start_Preheat;
   IF #_w1 AND NOT #State.Temp_Preheat_OK THEN #State.HWT_Status := 1; END_IF;
   IF #_w1 AND #State.Temp_Preheat_OK THEN #State.HWT_Status := 2; END_IF;
   #_w2 := #alwaysON AND NOT #Cmd.HWT_Mode AND #Cmd.Start_Prosses;
   IF #_w2 AND NOT #State.Temp_Process_OK THEN #State.HWT_Status := 3; END_IF;
   IF #_w2 AND #State.Temp_Process_OK AND NOT #State.Ready_for_Mix THEN #State.HWT_Status := 4; END_IF;
   IF #_w2 AND #State.Temp_Process_OK AND #State.Ready_for_Mix THEN #State.HWT_Status := 5; END_IF;
END_REGION

REGION Network 18: Enable_WHT_Mode
   RUNG wire#powerrail
      I_Contact( #Cmd.Start_Prosses )
      I_Contact( #Cmd.Start_Preheat )
      Coil( #State.Enable_WHT_Mode )
   END_RUNG
   // the same network as SCL:
   #State.Enable_WHT_Mode := NOT #Cmd.Start_Prosses AND NOT #Cmd.Start_Preheat;
END_REGION

REGION Network 19: Line Flow Switch
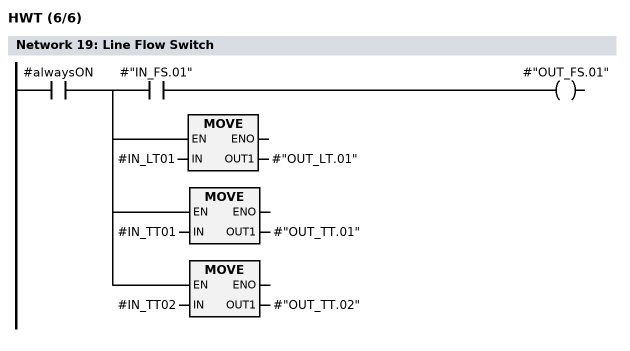
   RUNG wire#powerrail
      Contact( #alwaysON )
      wire#w1
      Contact( #"IN_FS.01" )
      Coil( #"OUT_FS.01" )
   END_RUNG
   RUNG wire#w1
      Move(in := #IN_LT01, out1 => #"OUT_LT.01")
   END_RUNG
   RUNG wire#w1
      Move(in := #IN_TT01, out1 => #"OUT_TT.01")
   END_RUNG
   RUNG wire#w1
      Move(in := #IN_TT02, out1 => #"OUT_TT.02")
   END_RUNG
   // the same network as SCL:
   #"OUT_FS.01" := #alwaysON AND #"IN_FS.01";
   IF #alwaysON THEN
       #"OUT_LT.01" := #IN_LT01;
       #"OUT_TT.01" := #IN_TT01;
       #"OUT_TT.02" := #IN_TT02;
   END_IF;
END_REGION
END_FUNCTION_BLOCK
